FUNCTION_BLOCK ST001_ProcessDataManager EXTENDS TcoData.TcoDataExchange
VAR
	_data : ST001_ProcessData;
END_VAR

SUPER^();

END_FUNCTION_BLOCK

(* stored: Version 1.1.0.1
   POU ST001_ProcessDataManager: Id {37e7eeae-cd25-0b59-3f07-4f9672bf8a09}, SpecialFunc None *)
